(* PLC project FiveDofPlatform_error_diag.import.xml, CODESYS CODESYS V3.5 SP20 Patch 4 *)
(* stored: creationDateTime 2026-08-01T11:31:50, modificationDateTime 2026-08-01T11:31:50 *)

PROGRAM AxisStatusFeedback_PRG
  VAR
    fbStatusX : Sm3_Basic.MC_ReadStatus;
    fbAxisErrorX : Sm3_Basic.MC_ReadAxisError;
    fbStatusY : Sm3_Basic.MC_ReadStatus;
    fbAxisErrorY : Sm3_Basic.MC_ReadAxisError;
    fbStatusZ : Sm3_Basic.MC_ReadStatus;
    fbAxisErrorZ : Sm3_Basic.MC_ReadAxisError;
    fbStatusB : Sm3_Basic.MC_ReadStatus;
    fbAxisErrorB : Sm3_Basic.MC_ReadAxisError;
    fbStatusC : Sm3_Basic.MC_ReadStatus;
    fbAxisErrorC : Sm3_Basic.MC_ReadAxisError;
    wStatusX : WORD;
    wStatusY : WORD;
    wStatusZ : WORD;
    wStatusB : WORD;
    wStatusC : WORD;
    dwAxisErrorX : DWORD;
    dwAxisErrorY : DWORD;
    dwAxisErrorZ : DWORD;
    dwAxisErrorB : DWORD;
    dwAxisErrorC : DWORD;
    bStatusErrorX : BOOL;
    bStatusFBErrorX : BOOL;
    bAxisErrorX : BOOL;
    bSwEndSwitchX : BOOL;
    bStatusErrorY : BOOL;
    bStatusFBErrorY : BOOL;
    bAxisErrorY : BOOL;
    bSwEndSwitchY : BOOL;
    bStatusErrorZ : BOOL;
    bStatusFBErrorZ : BOOL;
    bAxisErrorZ : BOOL;
    bSwEndSwitchZ : BOOL;
    bStatusErrorB : BOOL;
    bStatusFBErrorB : BOOL;
    bAxisErrorB : BOOL;
    bSwEndSwitchB : BOOL;
    bStatusErrorC : BOOL;
    bStatusFBErrorC : BOOL;
    bAxisErrorC : BOOL;
    bSwEndSwitchC : BOOL;
    eStatusErrorX : SMC_ERROR;
    eAxisReadErrorX : SMC_ERROR;
    bAxisReadErrorX : BOOL;
    eStatusErrorY : SMC_ERROR;
    eAxisReadErrorY : SMC_ERROR;
    bAxisReadErrorY : BOOL;
    eStatusErrorZ : SMC_ERROR;
    eAxisReadErrorZ : SMC_ERROR;
    bAxisReadErrorZ : BOOL;
    eStatusErrorB : SMC_ERROR;
    eAxisReadErrorB : SMC_ERROR;
    bAxisReadErrorB : BOOL;
    eStatusErrorC : SMC_ERROR;
    eAxisReadErrorC : SMC_ERROR;
    bAxisReadErrorC : BOOL;
    wEnableMismatchFeedback : WORD;
    wStatusErrorFeedback : WORD;
    wAxisReadErrorFeedback : WORD;
    wStatusFBErrorFeedback : WORD;
  END_VAR

            
// 本程序只做反馈和诊断，不直接控制轴运动。
// [32] 五轴总使能命令。
// [33..37] 五轴状态字。
// [38..47] 五轴驱动 AxisErrorID，来自 MC_ReadAxisError.AxisErrorID。
// [48] 五轴 AxisEnable 请求反馈。
// [49..58] 五轴 MC_ReadStatus.ErrorID。
// [59..68] 五轴 MC_ReadAxisError.ErrorID。
// [69..78] 五轴 MC_Power.ErrorID，由各单轴程序写入。
// [79..83] 五轴 MC_Power 诊断字，bit0=Status，bit1=Error。
// [84] 诊断版本号，26081 表示 2026-08-01 诊断版已生效。
// [85] 使能请求 TRUE 但 MC_ReadStatus 仍 Disabled 的位图。
// [86] MC_ReadStatus.Error 位图。
// [87] MC_ReadAxisError.Error 位图。
// [88] MC_ReadStatus.FBErrorOccured 位图。

fbStatusX(
    Axis := AXIS_X,
    Enable := TRUE,
    Valid => ,
    Busy => ,
    Error => bStatusErrorX,
    ErrorID => eStatusErrorX,
    Disabled => ,
    Errorstop => ,
    Stopping => ,
    StandStill => ,
    DiscreteMotion => ,
    ContinuousMotion => ,
    SynchronizedMotion => ,
    Homing => ,
    ConstantVelocity => ,
    Accelerating => ,
    Decelerating => ,
    FBErrorOccured => bStatusFBErrorX,
);

// MC_ReadAxisError.AxisErrorID 只表示驱动轴本体错误号。
// 如果网线断开导致 MC_ReadAxisError 自己报 Error，错误号会写到 arReg_data[59..60]。
fbAxisErrorX(
    Axis := AXIS_X,
    Enable := TRUE,
    Valid => ,
    Busy => ,
    Error => bAxisReadErrorX,
    ErrorID => eAxisReadErrorX,
    AxisError => bAxisErrorX,
    AxisErrorID => dwAxisErrorX,
    SWEndSwitchActive => bSwEndSwitchX
);
IF NOT bAxisErrorX THEN
    // 没有驱动轴本体错误时清零 AxisErrorID，但不清零各功能块自己的 ErrorID。
    dwAxisErrorX := DWORD#0;
END_IF;

// 把 X 轴 BOOL 状态压缩成一个 WORD 状态字输出到 arReg_data[33]。
wStatusX := WORD#0;
IF fbStatusX.Disabled THEN wStatusX := wStatusX OR WORD#16#0001; END_IF;
IF fbStatusX.Errorstop THEN wStatusX := wStatusX OR WORD#16#0002; END_IF;
IF fbStatusX.Stopping THEN wStatusX := wStatusX OR WORD#16#0004; END_IF;
IF fbStatusX.StandStill THEN wStatusX := wStatusX OR WORD#16#0008; END_IF;
IF fbStatusX.DiscreteMotion THEN wStatusX := wStatusX OR WORD#16#0010; END_IF;
IF fbStatusX.ContinuousMotion THEN wStatusX := wStatusX OR WORD#16#0020; END_IF;
IF fbStatusX.SynchronizedMotion THEN wStatusX := wStatusX OR WORD#16#0040; END_IF;
IF fbStatusX.Homing THEN wStatusX := wStatusX OR WORD#16#0080; END_IF;
IF fbStatusX.ConstantVelocity THEN wStatusX := wStatusX OR WORD#16#0100; END_IF;
IF fbStatusX.Accelerating THEN wStatusX := wStatusX OR WORD#16#0200; END_IF;
IF fbStatusX.Decelerating THEN wStatusX := wStatusX OR WORD#16#0400; END_IF;
IF bStatusErrorX THEN wStatusX := wStatusX OR WORD#16#0800; END_IF;
IF bStatusFBErrorX THEN wStatusX := wStatusX OR WORD#16#1000; END_IF;
IF bAxisErrorX THEN wStatusX := wStatusX OR WORD#16#4000; END_IF;
IF bSwEndSwitchX THEN wStatusX := wStatusX OR WORD#16#8000; END_IF;
arReg_data[33] := WORD_TO_INT(wStatusX);

// arReg_data[38..39] 保存 X 轴驱动 AxisErrorID。
arReg_data[38] := WORD_TO_INT(DWORD_TO_WORD(dwAxisErrorX));
arReg_data[39] := WORD_TO_INT(DWORD_TO_WORD(SHR(dwAxisErrorX, 16)));

// arReg_data[49..50] 保存 X 轴 MC_ReadStatus.ErrorID。
arReg_data[49] := WORD_TO_INT(DWORD_TO_WORD(TO_DWORD(eStatusErrorX)));
arReg_data[50] := WORD_TO_INT(DWORD_TO_WORD(SHR(TO_DWORD(eStatusErrorX), 16)));

// arReg_data[59..60] 保存 X 轴 MC_ReadAxisError.ErrorID。
arReg_data[59] := WORD_TO_INT(DWORD_TO_WORD(TO_DWORD(eAxisReadErrorX)));
arReg_data[60] := WORD_TO_INT(DWORD_TO_WORD(SHR(TO_DWORD(eAxisReadErrorX), 16)));

fbStatusY(
    Axis := AXIS_Y,
    Enable := TRUE,
    Valid => ,
    Busy => ,
    Error => bStatusErrorY,
    ErrorID => eStatusErrorY,
    Disabled => ,
    Errorstop => ,
    Stopping => ,
    StandStill => ,
    DiscreteMotion => ,
    ContinuousMotion => ,
    SynchronizedMotion => ,
    Homing => ,
    ConstantVelocity => ,
    Accelerating => ,
    Decelerating => ,
    FBErrorOccured => bStatusFBErrorY,
);

// MC_ReadAxisError.AxisErrorID 只表示驱动轴本体错误号。
// 如果网线断开导致 MC_ReadAxisError 自己报 Error，错误号会写到 arReg_data[61..62]。
fbAxisErrorY(
    Axis := AXIS_Y,
    Enable := TRUE,
    Valid => ,
    Busy => ,
    Error => bAxisReadErrorY,
    ErrorID => eAxisReadErrorY,
    AxisError => bAxisErrorY,
    AxisErrorID => dwAxisErrorY,
    SWEndSwitchActive => bSwEndSwitchY
);
IF NOT bAxisErrorY THEN
    // 没有驱动轴本体错误时清零 AxisErrorID，但不清零各功能块自己的 ErrorID。
    dwAxisErrorY := DWORD#0;
END_IF;

// 把 Y 轴 BOOL 状态压缩成一个 WORD 状态字输出到 arReg_data[34]。
wStatusY := WORD#0;
IF fbStatusY.Disabled THEN wStatusY := wStatusY OR WORD#16#0001; END_IF;
IF fbStatusY.Errorstop THEN wStatusY := wStatusY OR WORD#16#0002; END_IF;
IF fbStatusY.Stopping THEN wStatusY := wStatusY OR WORD#16#0004; END_IF;
IF fbStatusY.StandStill THEN wStatusY := wStatusY OR WORD#16#0008; END_IF;
IF fbStatusY.DiscreteMotion THEN wStatusY := wStatusY OR WORD#16#0010; END_IF;
IF fbStatusY.ContinuousMotion THEN wStatusY := wStatusY OR WORD#16#0020; END_IF;
IF fbStatusY.SynchronizedMotion THEN wStatusY := wStatusY OR WORD#16#0040; END_IF;
IF fbStatusY.Homing THEN wStatusY := wStatusY OR WORD#16#0080; END_IF;
IF fbStatusY.ConstantVelocity THEN wStatusY := wStatusY OR WORD#16#0100; END_IF;
IF fbStatusY.Accelerating THEN wStatusY := wStatusY OR WORD#16#0200; END_IF;
IF fbStatusY.Decelerating THEN wStatusY := wStatusY OR WORD#16#0400; END_IF;
IF bStatusErrorY THEN wStatusY := wStatusY OR WORD#16#0800; END_IF;
IF bStatusFBErrorY THEN wStatusY := wStatusY OR WORD#16#1000; END_IF;
IF bAxisErrorY THEN wStatusY := wStatusY OR WORD#16#4000; END_IF;
IF bSwEndSwitchY THEN wStatusY := wStatusY OR WORD#16#8000; END_IF;
arReg_data[34] := WORD_TO_INT(wStatusY);

// arReg_data[40..41] 保存 Y 轴驱动 AxisErrorID。
arReg_data[40] := WORD_TO_INT(DWORD_TO_WORD(dwAxisErrorY));
arReg_data[41] := WORD_TO_INT(DWORD_TO_WORD(SHR(dwAxisErrorY, 16)));

// arReg_data[51..52] 保存 Y 轴 MC_ReadStatus.ErrorID。
arReg_data[51] := WORD_TO_INT(DWORD_TO_WORD(TO_DWORD(eStatusErrorY)));
arReg_data[52] := WORD_TO_INT(DWORD_TO_WORD(SHR(TO_DWORD(eStatusErrorY), 16)));

// arReg_data[61..62] 保存 Y 轴 MC_ReadAxisError.ErrorID。
arReg_data[61] := WORD_TO_INT(DWORD_TO_WORD(TO_DWORD(eAxisReadErrorY)));
arReg_data[62] := WORD_TO_INT(DWORD_TO_WORD(SHR(TO_DWORD(eAxisReadErrorY), 16)));

fbStatusZ(
    Axis := AXIS_Z,
    Enable := TRUE,
    Valid => ,
    Busy => ,
    Error => bStatusErrorZ,
    ErrorID => eStatusErrorZ,
    Disabled => ,
    Errorstop => ,
    Stopping => ,
    StandStill => ,
    DiscreteMotion => ,
    ContinuousMotion => ,
    SynchronizedMotion => ,
    Homing => ,
    ConstantVelocity => ,
    Accelerating => ,
    Decelerating => ,
    FBErrorOccured => bStatusFBErrorZ,
);

// MC_ReadAxisError.AxisErrorID 只表示驱动轴本体错误号。
// 如果网线断开导致 MC_ReadAxisError 自己报 Error，错误号会写到 arReg_data[63..64]。
fbAxisErrorZ(
    Axis := AXIS_Z,
    Enable := TRUE,
    Valid => ,
    Busy => ,
    Error => bAxisReadErrorZ,
    ErrorID => eAxisReadErrorZ,
    AxisError => bAxisErrorZ,
    AxisErrorID => dwAxisErrorZ,
    SWEndSwitchActive => bSwEndSwitchZ
);
IF NOT bAxisErrorZ THEN
    // 没有驱动轴本体错误时清零 AxisErrorID，但不清零各功能块自己的 ErrorID。
    dwAxisErrorZ := DWORD#0;
END_IF;

// 把 Z 轴 BOOL 状态压缩成一个 WORD 状态字输出到 arReg_data[35]。
wStatusZ := WORD#0;
IF fbStatusZ.Disabled THEN wStatusZ := wStatusZ OR WORD#16#0001; END_IF;
IF fbStatusZ.Errorstop THEN wStatusZ := wStatusZ OR WORD#16#0002; END_IF;
IF fbStatusZ.Stopping THEN wStatusZ := wStatusZ OR WORD#16#0004; END_IF;
IF fbStatusZ.StandStill THEN wStatusZ := wStatusZ OR WORD#16#0008; END_IF;
IF fbStatusZ.DiscreteMotion THEN wStatusZ := wStatusZ OR WORD#16#0010; END_IF;
IF fbStatusZ.ContinuousMotion THEN wStatusZ := wStatusZ OR WORD#16#0020; END_IF;
IF fbStatusZ.SynchronizedMotion THEN wStatusZ := wStatusZ OR WORD#16#0040; END_IF;
IF fbStatusZ.Homing THEN wStatusZ := wStatusZ OR WORD#16#0080; END_IF;
IF fbStatusZ.ConstantVelocity THEN wStatusZ := wStatusZ OR WORD#16#0100; END_IF;
IF fbStatusZ.Accelerating THEN wStatusZ := wStatusZ OR WORD#16#0200; END_IF;
IF fbStatusZ.Decelerating THEN wStatusZ := wStatusZ OR WORD#16#0400; END_IF;
IF bStatusErrorZ THEN wStatusZ := wStatusZ OR WORD#16#0800; END_IF;
IF bStatusFBErrorZ THEN wStatusZ := wStatusZ OR WORD#16#1000; END_IF;
IF bAxisErrorZ THEN wStatusZ := wStatusZ OR WORD#16#4000; END_IF;
IF bSwEndSwitchZ THEN wStatusZ := wStatusZ OR WORD#16#8000; END_IF;
arReg_data[35] := WORD_TO_INT(wStatusZ);

// arReg_data[42..43] 保存 Z 轴驱动 AxisErrorID。
arReg_data[42] := WORD_TO_INT(DWORD_TO_WORD(dwAxisErrorZ));
arReg_data[43] := WORD_TO_INT(DWORD_TO_WORD(SHR(dwAxisErrorZ, 16)));

// arReg_data[53..54] 保存 Z 轴 MC_ReadStatus.ErrorID。
arReg_data[53] := WORD_TO_INT(DWORD_TO_WORD(TO_DWORD(eStatusErrorZ)));
arReg_data[54] := WORD_TO_INT(DWORD_TO_WORD(SHR(TO_DWORD(eStatusErrorZ), 16)));

// arReg_data[63..64] 保存 Z 轴 MC_ReadAxisError.ErrorID。
arReg_data[63] := WORD_TO_INT(DWORD_TO_WORD(TO_DWORD(eAxisReadErrorZ)));
arReg_data[64] := WORD_TO_INT(DWORD_TO_WORD(SHR(TO_DWORD(eAxisReadErrorZ), 16)));

fbStatusB(
    Axis := AXIS_B,
    Enable := TRUE,
    Valid => ,
    Busy => ,
    Error => bStatusErrorB,
    ErrorID => eStatusErrorB,
    Disabled => ,
    Errorstop => ,
    Stopping => ,
    StandStill => ,
    DiscreteMotion => ,
    ContinuousMotion => ,
    SynchronizedMotion => ,
    Homing => ,
    ConstantVelocity => ,
    Accelerating => ,
    Decelerating => ,
    FBErrorOccured => bStatusFBErrorB,
);

// MC_ReadAxisError.AxisErrorID 只表示驱动轴本体错误号。
// 如果网线断开导致 MC_ReadAxisError 自己报 Error，错误号会写到 arReg_data[65..66]。
fbAxisErrorB(
    Axis := AXIS_B,
    Enable := TRUE,
    Valid => ,
    Busy => ,
    Error => bAxisReadErrorB,
    ErrorID => eAxisReadErrorB,
    AxisError => bAxisErrorB,
    AxisErrorID => dwAxisErrorB,
    SWEndSwitchActive => bSwEndSwitchB
);
IF NOT bAxisErrorB THEN
    // 没有驱动轴本体错误时清零 AxisErrorID，但不清零各功能块自己的 ErrorID。
    dwAxisErrorB := DWORD#0;
END_IF;

// 把 B 轴 BOOL 状态压缩成一个 WORD 状态字输出到 arReg_data[36]。
wStatusB := WORD#0;
IF fbStatusB.Disabled THEN wStatusB := wStatusB OR WORD#16#0001; END_IF;
IF fbStatusB.Errorstop THEN wStatusB := wStatusB OR WORD#16#0002; END_IF;
IF fbStatusB.Stopping THEN wStatusB := wStatusB OR WORD#16#0004; END_IF;
IF fbStatusB.StandStill THEN wStatusB := wStatusB OR WORD#16#0008; END_IF;
IF fbStatusB.DiscreteMotion THEN wStatusB := wStatusB OR WORD#16#0010; END_IF;
IF fbStatusB.ContinuousMotion THEN wStatusB := wStatusB OR WORD#16#0020; END_IF;
IF fbStatusB.SynchronizedMotion THEN wStatusB := wStatusB OR WORD#16#0040; END_IF;
IF fbStatusB.Homing THEN wStatusB := wStatusB OR WORD#16#0080; END_IF;
IF fbStatusB.ConstantVelocity THEN wStatusB := wStatusB OR WORD#16#0100; END_IF;
IF fbStatusB.Accelerating THEN wStatusB := wStatusB OR WORD#16#0200; END_IF;
IF fbStatusB.Decelerating THEN wStatusB := wStatusB OR WORD#16#0400; END_IF;
IF bStatusErrorB THEN wStatusB := wStatusB OR WORD#16#0800; END_IF;
IF bStatusFBErrorB THEN wStatusB := wStatusB OR WORD#16#1000; END_IF;
IF bAxisErrorB THEN wStatusB := wStatusB OR WORD#16#4000; END_IF;
IF bSwEndSwitchB THEN wStatusB := wStatusB OR WORD#16#8000; END_IF;
arReg_data[36] := WORD_TO_INT(wStatusB);

// arReg_data[44..45] 保存 B 轴驱动 AxisErrorID。
arReg_data[44] := WORD_TO_INT(DWORD_TO_WORD(dwAxisErrorB));
arReg_data[45] := WORD_TO_INT(DWORD_TO_WORD(SHR(dwAxisErrorB, 16)));

// arReg_data[55..56] 保存 B 轴 MC_ReadStatus.ErrorID。
arReg_data[55] := WORD_TO_INT(DWORD_TO_WORD(TO_DWORD(eStatusErrorB)));
arReg_data[56] := WORD_TO_INT(DWORD_TO_WORD(SHR(TO_DWORD(eStatusErrorB), 16)));

// arReg_data[65..66] 保存 B 轴 MC_ReadAxisError.ErrorID。
arReg_data[65] := WORD_TO_INT(DWORD_TO_WORD(TO_DWORD(eAxisReadErrorB)));
arReg_data[66] := WORD_TO_INT(DWORD_TO_WORD(SHR(TO_DWORD(eAxisReadErrorB), 16)));

fbStatusC(
    Axis := AXIS_C,
    Enable := TRUE,
    Valid => ,
    Busy => ,
    Error => bStatusErrorC,
    ErrorID => eStatusErrorC,
    Disabled => ,
    Errorstop => ,
    Stopping => ,
    StandStill => ,
    DiscreteMotion => ,
    ContinuousMotion => ,
    SynchronizedMotion => ,
    Homing => ,
    ConstantVelocity => ,
    Accelerating => ,
    Decelerating => ,
    FBErrorOccured => bStatusFBErrorC,
);

// MC_ReadAxisError.AxisErrorID 只表示驱动轴本体错误号。
// 如果网线断开导致 MC_ReadAxisError 自己报 Error，错误号会写到 arReg_data[67..68]。
fbAxisErrorC(
    Axis := AXIS_C,
    Enable := TRUE,
    Valid => ,
    Busy => ,
    Error => bAxisReadErrorC,
    ErrorID => eAxisReadErrorC,
    AxisError => bAxisErrorC,
    AxisErrorID => dwAxisErrorC,
    SWEndSwitchActive => bSwEndSwitchC
);
IF NOT bAxisErrorC THEN
    // 没有驱动轴本体错误时清零 AxisErrorID，但不清零各功能块自己的 ErrorID。
    dwAxisErrorC := DWORD#0;
END_IF;

// 把 C 轴 BOOL 状态压缩成一个 WORD 状态字输出到 arReg_data[37]。
wStatusC := WORD#0;
IF fbStatusC.Disabled THEN wStatusC := wStatusC OR WORD#16#0001; END_IF;
IF fbStatusC.Errorstop THEN wStatusC := wStatusC OR WORD#16#0002; END_IF;
IF fbStatusC.Stopping THEN wStatusC := wStatusC OR WORD#16#0004; END_IF;
IF fbStatusC.StandStill THEN wStatusC := wStatusC OR WORD#16#0008; END_IF;
IF fbStatusC.DiscreteMotion THEN wStatusC := wStatusC OR WORD#16#0010; END_IF;
IF fbStatusC.ContinuousMotion THEN wStatusC := wStatusC OR WORD#16#0020; END_IF;
IF fbStatusC.SynchronizedMotion THEN wStatusC := wStatusC OR WORD#16#0040; END_IF;
IF fbStatusC.Homing THEN wStatusC := wStatusC OR WORD#16#0080; END_IF;
IF fbStatusC.ConstantVelocity THEN wStatusC := wStatusC OR WORD#16#0100; END_IF;
IF fbStatusC.Accelerating THEN wStatusC := wStatusC OR WORD#16#0200; END_IF;
IF fbStatusC.Decelerating THEN wStatusC := wStatusC OR WORD#16#0400; END_IF;
IF bStatusErrorC THEN wStatusC := wStatusC OR WORD#16#0800; END_IF;
IF bStatusFBErrorC THEN wStatusC := wStatusC OR WORD#16#1000; END_IF;
IF bAxisErrorC THEN wStatusC := wStatusC OR WORD#16#4000; END_IF;
IF bSwEndSwitchC THEN wStatusC := wStatusC OR WORD#16#8000; END_IF;
arReg_data[37] := WORD_TO_INT(wStatusC);

// arReg_data[46..47] 保存 C 轴驱动 AxisErrorID。
arReg_data[46] := WORD_TO_INT(DWORD_TO_WORD(dwAxisErrorC));
arReg_data[47] := WORD_TO_INT(DWORD_TO_WORD(SHR(dwAxisErrorC, 16)));

// arReg_data[57..58] 保存 C 轴 MC_ReadStatus.ErrorID。
arReg_data[57] := WORD_TO_INT(DWORD_TO_WORD(TO_DWORD(eStatusErrorC)));
arReg_data[58] := WORD_TO_INT(DWORD_TO_WORD(SHR(TO_DWORD(eStatusErrorC), 16)));

// arReg_data[67..68] 保存 C 轴 MC_ReadAxisError.ErrorID。
arReg_data[67] := WORD_TO_INT(DWORD_TO_WORD(TO_DWORD(eAxisReadErrorC)));
arReg_data[68] := WORD_TO_INT(DWORD_TO_WORD(SHR(TO_DWORD(eAxisReadErrorC), 16)));

// 诊断版本号，Python 可用它判断 [49..88] 是否已由新版 PLC 代码写入。
arReg_data[84] := 26081;

// 使能请求不一致：AxisEnable 请求为 TRUE，但 MC_ReadStatus 仍显示 Disabled。
wEnableMismatchFeedback := WORD#0;
IF GVL.Axes[1].AxisEnable AND fbStatusX.Disabled THEN wEnableMismatchFeedback := wEnableMismatchFeedback OR WORD#16#0001; END_IF;
IF GVL.Axes[2].AxisEnable AND fbStatusY.Disabled THEN wEnableMismatchFeedback := wEnableMismatchFeedback OR WORD#16#0002; END_IF;
IF GVL.Axes[3].AxisEnable AND fbStatusZ.Disabled THEN wEnableMismatchFeedback := wEnableMismatchFeedback OR WORD#16#0004; END_IF;
IF GVL.Axes[4].AxisEnable AND fbStatusB.Disabled THEN wEnableMismatchFeedback := wEnableMismatchFeedback OR WORD#16#0008; END_IF;
IF GVL.Axes[5].AxisEnable AND fbStatusC.Disabled THEN wEnableMismatchFeedback := wEnableMismatchFeedback OR WORD#16#0010; END_IF;
arReg_data[85] := WORD_TO_INT(wEnableMismatchFeedback);

// 汇总功能块错误位，便于 Python 快速判断是哪一类诊断报错。
wStatusErrorFeedback := WORD#0;
IF bStatusErrorX THEN wStatusErrorFeedback := wStatusErrorFeedback OR WORD#16#0001; END_IF;
IF bStatusErrorY THEN wStatusErrorFeedback := wStatusErrorFeedback OR WORD#16#0002; END_IF;
IF bStatusErrorZ THEN wStatusErrorFeedback := wStatusErrorFeedback OR WORD#16#0004; END_IF;
IF bStatusErrorB THEN wStatusErrorFeedback := wStatusErrorFeedback OR WORD#16#0008; END_IF;
IF bStatusErrorC THEN wStatusErrorFeedback := wStatusErrorFeedback OR WORD#16#0010; END_IF;
arReg_data[86] := WORD_TO_INT(wStatusErrorFeedback);

wAxisReadErrorFeedback := WORD#0;
IF bAxisReadErrorX THEN wAxisReadErrorFeedback := wAxisReadErrorFeedback OR WORD#16#0001; END_IF;
IF bAxisReadErrorY THEN wAxisReadErrorFeedback := wAxisReadErrorFeedback OR WORD#16#0002; END_IF;
IF bAxisReadErrorZ THEN wAxisReadErrorFeedback := wAxisReadErrorFeedback OR WORD#16#0004; END_IF;
IF bAxisReadErrorB THEN wAxisReadErrorFeedback := wAxisReadErrorFeedback OR WORD#16#0008; END_IF;
IF bAxisReadErrorC THEN wAxisReadErrorFeedback := wAxisReadErrorFeedback OR WORD#16#0010; END_IF;
arReg_data[87] := WORD_TO_INT(wAxisReadErrorFeedback);

wStatusFBErrorFeedback := WORD#0;
IF bStatusFBErrorX THEN wStatusFBErrorFeedback := wStatusFBErrorFeedback OR WORD#16#0001; END_IF;
IF bStatusFBErrorY THEN wStatusFBErrorFeedback := wStatusFBErrorFeedback OR WORD#16#0002; END_IF;
IF bStatusFBErrorZ THEN wStatusFBErrorFeedback := wStatusFBErrorFeedback OR WORD#16#0004; END_IF;
IF bStatusFBErrorB THEN wStatusFBErrorFeedback := wStatusFBErrorFeedback OR WORD#16#0008; END_IF;
IF bStatusFBErrorC THEN wStatusFBErrorFeedback := wStatusFBErrorFeedback OR WORD#16#0010; END_IF;
arReg_data[88] := WORD_TO_INT(wStatusFBErrorFeedback);

          
END_PROGRAM

PROGRAM AXIS_X_PRG
  VAR
    伺服使能 : Sm3_Basic.MC_Power;  (* 轴功能块实例 *)
    伺服绝对位置执行 : Sm3_Basic.MC_MoveAbsolute;
    伺服实际位置 : Sm3_Basic.MC_ReadActualPosition;
    伺服停止 : Sm3_Basic.MC_Stop;
    伺服复位 : Sm3_Basic.MC_Reset;
    伺服状态 : Sm3_Basic.MC_ReadStatus;
    复位轴组 : Sm3_Basic.SMC3_ReinitDrive;
    当前位置 : LREAL;  (* 变量 *)
    轴组复位 : BOOL;
    目标位置 : LREAL;
    目标速度 : LREAL;
    伺服错误状态 : BOOL;
    轴使能状态 : BOOL;
    总线状态 : BOOL;
    复位触发 : R_TRIG;  (* 报警清除相关 *)
    复位请求 : BOOL;
    复位中 : BOOL;
    POS_DEAD_ZONE : REAL := 0.01;  (* 死区常量 *)
    move_trigger : R_TRIG;
    AXIS_X_EXCUSE : BOOL := FALSE;
    log_msg : STRING(100);
    bPowerErrorDiag : BOOL;
    ePowerErrorDiag : SMC_ERROR;
    wPowerDiag : WORD;
  END_VAR

                    //------------------------------------------------------------------
// Z 轴控制逻辑（简化版 - 仅上升沿触发）
//------------------------------------------------------------------

// 读取实际位置
伺服实际位置(
    Axis    := AXIS_X,
    Enable  := TRUE,
    Position=> 当前位置
);
GVL.Axes[1].ActualAngle := 当前位置;

// 读取轴状态
伺服状态(
    Axis    := AXIS_X,
    Enable  := TRUE,
    Valid   => ,
    Busy    => ,
    Error   => 伺服错误状态,
    ErrorID => ,
    Disabled=> 总线状态
);

// 轴使能控制
伺服使能(
    Axis               := AXIS_X,
    Enable             := TRUE,
    bRegulatorOn       := GVL.Axes[1].AxisEnable,
    bDriveStart        := GVL.Axes[1].AxisEnable,
    Status             => 轴使能状态,
    bRegulatorRealState=> ,
    bDriveStartRealState=> ,
    Busy               => ,
    Error              => bPowerErrorDiag,
    ErrorID            => ePowerErrorDiag
);


// arReg_data[69..70] 保存本轴 MC_Power.ErrorID。
// 拔网线、驱动掉线、电机线导致的上使能故障，常先从这里体现。
arReg_data[69] := WORD_TO_INT(DWORD_TO_WORD(TO_DWORD(ePowerErrorDiag)));
arReg_data[70] := WORD_TO_INT(DWORD_TO_WORD(SHR(TO_DWORD(ePowerErrorDiag), 16)));

// arReg_data[79] 保存本轴 MC_Power 诊断字：bit0=Status，bit1=Error。
wPowerDiag := WORD#0;
IF 轴使能状态 THEN wPowerDiag := wPowerDiag OR WORD#16#0001; END_IF;
IF bPowerErrorDiag THEN wPowerDiag := wPowerDiag OR WORD#16#0002; END_IF;
arReg_data[79] := WORD_TO_INT(wPowerDiag);

// 目标位置、速度赋值（来自全局变量）
目标位置 := GVL.Axes[1].TargetAngle;
目标速度 :=  GVL.Axes[1].TargetVel;

// ********** 核心：上升沿触发运动 **********
// 使用 R_TRIG 检测 need_move 的上升沿
move_trigger(CLK := GVL.Axes[1].NeedMoveAxis);
IF move_trigger.Q THEN
    AXIS_X_EXCUSE := TRUE;   // 产生一个扫描周期的脉冲
	log_msg := 'X-axis has been triggered';
// 	logfb(write:=TRUE,sFileTestString:=log_msg);
	AppendLog(log_msg);
ELSE
    AXIS_X_EXCUSE := FALSE;
END_IF

// 绝对定位指令
GVL.Axes[1].伺服绝对位置执行(
    Axis        := AXIS_X,
    Execute     := AXIS_X_EXCUSE,
    Position    := 目标位置,
    Velocity    := 目标速度,
    Acceleration:= 10000,//4000  //85000
    Deceleration:= 10000,//4000  //85000
    Jerk        := ,
    Direction   := ,
    BufferMode  := ,
    Done        => GVL.Axes[1].InitDone,
    Busy        => ,
    Active      => ,
    CommandAborted=> ,
    Error       => GVL.Axes[1].AxisError,
    ErrorID     =>
);

// 运动完成：清除 need_move 并通知状态机
IF  GVL.Axes[1].InitDone THEN
    GVL.Axes[1].NeedMoveAxis := FALSE;              // 清除运动请求
    GVL.Axes[1].AxisDone := TRUE;         // 通知状态机运动完成
	log_msg := 'X-Axis movement completed! ';
// 	logfb(write:=TRUE,sFileTestString:=log_msg);
// 	AppendLog(log_msg);
END_IF

// 复位功能块（保持不变）
伺服复位(
    Axis    := AXIS_X,
    Execute := 复位中 AND NOT 伺服复位.Done,
    Done    => ,
    Busy    => ,
    Error   => ,
    ErrorID =>
);

复位轴组(
    Axis      := AXIS_X,
    bExecute  := 伺服复位.Done,
    bVirtual  := FALSE,
    bDone     => ,
    bBusy     => ,
    bError    => ,
    nErrorID  =>
);

// 报警清除逻辑
复位触发(CLK := (伺服错误状态 OR 复位请求) AND NOT 复位中);
IF 复位触发.Q THEN
    复位中 := TRUE;
    复位请求 := FALSE;
END_IF

IF 伺服复位.Done THEN
    复位中 := FALSE;
END_IF
                  
END_PROGRAM

PROGRAM Axis_Y_PRG
  VAR
    伺服使能 : Sm3_Basic.MC_Power;  (* 轴功能块实例 *)
    伺服绝对位置执行 : Sm3_Basic.MC_MoveAbsolute;
    伺服实际位置 : Sm3_Basic.MC_ReadActualPosition;
    伺服停止 : Sm3_Basic.MC_Stop;
    伺服复位 : Sm3_Basic.MC_Reset;
    伺服状态 : Sm3_Basic.MC_ReadStatus;
    复位轴组 : Sm3_Basic.SMC3_ReinitDrive;
    当前位置 : LREAL;  (* 变量 *)
    轴组复位 : BOOL;
    目标位置 : LREAL;
    目标速度 : LREAL;
    伺服错误状态 : BOOL;
    轴使能状态 : BOOL;
    总线状态 : BOOL;
    复位触发 : R_TRIG;  (* 报警清除相关 *)
    复位请求 : BOOL;
    复位中 : BOOL;
    POS_DEAD_ZONE : REAL := 0.01;  (* 死区常量 *)
    伺服复位_Done : BOOL;
    debug_Done_Status : BOOL;  (* 在 AXIS_Y0_PRG 中添加 *)
    debug_KeepEnable : BOOL;
    move_trigger : R_TRIG;  (* 脉冲触发相关 *)
    AXIS_Y_EXCUSE : BOOL := FALSE;
    log_msg : STRING(100);
    bPowerErrorDiag : BOOL;
    ePowerErrorDiag : SMC_ERROR;
    wPowerDiag : WORD;
  END_VAR

                    //------------------------------------------------------------------
// Z 轴控制逻辑（简化版 - 仅上升沿触发）
//------------------------------------------------------------------

// 读取实际位置
伺服实际位置(
    Axis    := AXIS_Y,
    Enable  := TRUE,
    Position=> 当前位置
);
GVL.Axes[2].ActualAngle := 当前位置;

// 读取轴状态
伺服状态(
    Axis    := AXIS_Y,
    Enable  := TRUE,
    Valid   => ,
    Busy    => ,
    Error   => 伺服错误状态,
    ErrorID => ,
    Disabled=> 总线状态
);

// 轴使能控制
伺服使能(
    Axis               := AXIS_Y,
    Enable             := TRUE,
    bRegulatorOn       := GVL.Axes[2].AxisEnable,
    bDriveStart        := GVL.Axes[2].AxisEnable,
    Status             => 轴使能状态,
    bRegulatorRealState=> ,
    bDriveStartRealState=> ,
    Busy               => ,
    Error              => bPowerErrorDiag,
    ErrorID            => ePowerErrorDiag
);


// arReg_data[71..72] 保存本轴 MC_Power.ErrorID。
// 拔网线、驱动掉线、电机线导致的上使能故障，常先从这里体现。
arReg_data[71] := WORD_TO_INT(DWORD_TO_WORD(TO_DWORD(ePowerErrorDiag)));
arReg_data[72] := WORD_TO_INT(DWORD_TO_WORD(SHR(TO_DWORD(ePowerErrorDiag), 16)));

// arReg_data[80] 保存本轴 MC_Power 诊断字：bit0=Status，bit1=Error。
wPowerDiag := WORD#0;
IF 轴使能状态 THEN wPowerDiag := wPowerDiag OR WORD#16#0001; END_IF;
IF bPowerErrorDiag THEN wPowerDiag := wPowerDiag OR WORD#16#0002; END_IF;
arReg_data[80] := WORD_TO_INT(wPowerDiag);

// 目标位置、速度赋值（来自全局变量）
目标位置 := GVL.Axes[2].TargetAngle;
目标速度 :=  GVL.Axes[2].TargetVel;

// ********** 核心：上升沿触发运动 **********
// 使用 R_TRIG 检测 need_move 的上升沿
move_trigger(CLK := GVL.Axes[2].NeedMoveAxis);
IF move_trigger.Q THEN
    AXIS_Y_EXCUSE := TRUE;   // 产生一个扫描周期的脉冲
	log_msg := 'X-axis has been triggered';
// 	logfb(write:=TRUE,sFileTestString:=log_msg);
	AppendLog(log_msg);
ELSE
    AXIS_Y_EXCUSE := FALSE;
END_IF

// 绝对定位指令
GVL.Axes[2].伺服绝对位置执行(
    Axis        := AXIS_Y,
    Execute     := AXIS_Y_EXCUSE,
    Position    := 目标位置,
    Velocity    := 目标速度,
    Acceleration:= 10000,//4000  //85000
    Deceleration:= 10000,//4000  //85000
    Jerk        := ,
    Direction   := ,
    BufferMode  := ,
    Done        => GVL.Axes[2].InitDone,
    Busy        => ,
    Active      => ,
    CommandAborted=> ,
    Error       => GVL.Axes[2].AxisError,
    ErrorID     =>
);

// 运动完成：清除 need_move 并通知状态机
IF  GVL.Axes[2].InitDone THEN
    GVL.Axes[2].NeedMoveAxis := FALSE;              // 清除运动请求
    GVL.Axes[2].AxisDone := TRUE;         // 通知状态机运动完成
	log_msg := 'X-Axis movement completed! ';
// 	logfb(write:=TRUE,sFileTestString:=log_msg);
// 	AppendLog(log_msg);
END_IF

// 复位功能块（保持不变）
伺服复位(
    Axis    := AXIS_Y,
    Execute := 复位中 AND NOT 伺服复位.Done,
    Done    => ,
    Busy    => ,
    Error   => ,
    ErrorID =>
);

复位轴组(
    Axis      := AXIS_Y,
    bExecute  := 伺服复位.Done,
    bVirtual  := FALSE,
    bDone     => ,
    bBusy     => ,
    bError    => ,
    nErrorID  =>
);

// 报警清除逻辑
复位触发(CLK := (伺服错误状态 OR 复位请求) AND NOT 复位中);
IF 复位触发.Q THEN
    复位中 := TRUE;
    复位请求 := FALSE;
END_IF

IF 伺服复位.Done THEN
    复位中 := FALSE;
END_IF
                  
END_PROGRAM

PROGRAM AXIS_Z_PRG
  VAR
    伺服使能 : Sm3_Basic.MC_Power;  (* 轴功能块实例 *)
    伺服绝对位置执行 : Sm3_Basic.MC_MoveAbsolute;
    伺服实际位置 : Sm3_Basic.MC_ReadActualPosition;
    伺服停止 : Sm3_Basic.MC_Stop;
    伺服复位 : Sm3_Basic.MC_Reset;
    伺服状态 : Sm3_Basic.MC_ReadStatus;
    复位轴组 : Sm3_Basic.SMC3_ReinitDrive;
    当前位置 : LREAL;  (* 变量 *)
    轴组复位 : BOOL;
    目标位置 : LREAL;
    目标速度 : LREAL;
    伺服错误状态 : BOOL;
    轴使能状态 : BOOL;
    总线状态 : BOOL;
    复位触发 : R_TRIG;  (* 报警清除相关 *)
    复位请求 : BOOL;
    复位中 : BOOL;
    伺服复位_Done : BOOL;
    debug_Done_Status : BOOL;  (* 在 AXIS_Z_PRG 中添加 *)
    debug_KeepEnable : BOOL;
    move_trigger : R_TRIG;  (* 脉冲触发相关 *)
    AXIS_Z_EXCUSE : BOOL := FALSE;
    log_msg : STRING(100);
    bPowerErrorDiag : BOOL;
    ePowerErrorDiag : SMC_ERROR;
    wPowerDiag : WORD;
  END_VAR

                    //------------------------------------------------------------------
// Z 轴控制逻辑（简化版 - 仅上升沿触发）
//------------------------------------------------------------------

// 读取实际位置
伺服实际位置(
    Axis    := AXIS_Z,
    Enable  := TRUE,
    Position=> 当前位置
);
GVL.Axes[3].ActualAngle := 当前位置;

// 读取轴状态
伺服状态(
    Axis    := AXIS_Z,
    Enable  := TRUE,
    Valid   => ,
    Busy    => ,
    Error   => 伺服错误状态,
    ErrorID => ,
    Disabled=> 总线状态
);

// 轴使能控制
伺服使能(
    Axis               := AXIS_Z,
    Enable             := TRUE,
    bRegulatorOn       := GVL.Axes[3].AxisEnable,
    bDriveStart        := GVL.Axes[3].AxisEnable,
    Status             => 轴使能状态,
    bRegulatorRealState=> ,
    bDriveStartRealState=> ,
    Busy               => ,
    Error              => bPowerErrorDiag,
    ErrorID            => ePowerErrorDiag
);


// arReg_data[73..74] 保存本轴 MC_Power.ErrorID。
// 拔网线、驱动掉线、电机线导致的上使能故障，常先从这里体现。
arReg_data[73] := WORD_TO_INT(DWORD_TO_WORD(TO_DWORD(ePowerErrorDiag)));
arReg_data[74] := WORD_TO_INT(DWORD_TO_WORD(SHR(TO_DWORD(ePowerErrorDiag), 16)));

// arReg_data[81] 保存本轴 MC_Power 诊断字：bit0=Status，bit1=Error。
wPowerDiag := WORD#0;
IF 轴使能状态 THEN wPowerDiag := wPowerDiag OR WORD#16#0001; END_IF;
IF bPowerErrorDiag THEN wPowerDiag := wPowerDiag OR WORD#16#0002; END_IF;
arReg_data[81] := WORD_TO_INT(wPowerDiag);

// 目标位置、速度赋值（来自全局变量）
目标位置 := GVL.Axes[3].TargetAngle;
目标速度 :=  GVL.Axes[3].TargetVel;

// ********** 核心：上升沿触发运动 **********
// 使用 R_TRIG 检测 need_move 的上升沿
move_trigger(CLK := GVL.Axes[3].NeedMoveAxis);
IF move_trigger.Q THEN
    AXIS_Z_EXCUSE := TRUE;   // 产生一个扫描周期的脉冲
	log_msg := 'X-axis has been triggered';
// 	logfb(write:=TRUE,sFileTestString:=log_msg);
	AppendLog(log_msg);
ELSE
    AXIS_Z_EXCUSE := FALSE;
END_IF

// 绝对定位指令
GVL.Axes[3].伺服绝对位置执行(
    Axis        := AXIS_Z,
    Execute     := AXIS_Z_EXCUSE,
    Position    := 目标位置,
    Velocity    := 目标速度,
    Acceleration:= 10000,//4000  //85000
    Deceleration:= 10000,//4000  //85000
    Jerk        := ,
    Direction   := ,
    BufferMode  := ,
    Done        => GVL.Axes[3].InitDone,
    Busy        => ,
    Active      => ,
    CommandAborted=> ,
    Error       => GVL.Axes[3].AxisError,
    ErrorID     =>
);

// 运动完成：清除 need_move 并通知状态机
IF  GVL.Axes[3].InitDone THEN
    GVL.Axes[3].NeedMoveAxis := FALSE;              // 清除运动请求
    GVL.Axes[3].AxisDone := TRUE;         // 通知状态机运动完成
	log_msg := 'Z-Axis movement completed! ';
// 	logfb(write:=TRUE,sFileTestString:=log_msg);
// 	AppendLog(log_msg);
END_IF

// 复位功能块（保持不变）
伺服复位(
    Axis    := AXIS_Z,
    Execute := 复位中 AND NOT 伺服复位.Done,
    Done    => ,
    Busy    => ,
    Error   => ,
    ErrorID =>
);

复位轴组(
    Axis      := AXIS_Z,
    bExecute  := 伺服复位.Done,
    bVirtual  := FALSE,
    bDone     => ,
    bBusy     => ,
    bError    => ,
    nErrorID  =>
);

// 报警清除逻辑
复位触发(CLK := (伺服错误状态 OR 复位请求) AND NOT 复位中);
IF 复位触发.Q THEN
    复位中 := TRUE;
    复位请求 := FALSE;
END_IF

IF 伺服复位.Done THEN
    复位中 := FALSE;
END_IF
                  
END_PROGRAM

PROGRAM AXIS_B_PRG
  VAR
    伺服使能 : Sm3_Basic.MC_Power;  (* 轴功能块实例 *)
    伺服绝对位置执行 : Sm3_Basic.MC_MoveAbsolute;
    伺服实际位置 : Sm3_Basic.MC_ReadActualPosition;
    伺服停止 : Sm3_Basic.MC_Stop;
    伺服复位 : Sm3_Basic.MC_Reset;
    伺服状态 : Sm3_Basic.MC_ReadStatus;
    复位轴组 : Sm3_Basic.SMC3_ReinitDrive;
    当前位置 : LREAL;  (* 变量 *)
    轴组复位 : BOOL;
    目标位置 : LREAL;
    目标速度 : LREAL;
    伺服错误状态 : BOOL;
    轴使能状态 : BOOL;
    总线状态 : BOOL;
    复位触发 : R_TRIG;  (* 报警清除相关 *)
    复位请求 : BOOL;
    复位中 : BOOL;
    move_trigger : R_TRIG;
    AXIS_B_EXCUSE : BOOL := FALSE;
    log_msg : STRING(100);
    bPowerErrorDiag : BOOL;
    ePowerErrorDiag : SMC_ERROR;
    wPowerDiag : WORD;
  END_VAR

                    //------------------------------------------------------------------
// Z 轴控制逻辑（简化版 - 仅上升沿触发）
//------------------------------------------------------------------

// 读取实际位置
伺服实际位置(
    Axis    := AXIS_B,
    Enable  := TRUE,
    Position=> 当前位置
);
GVL.Axes[4].ActualAngle := 当前位置;

// 读取轴状态
伺服状态(
    Axis    := AXIS_B,
    Enable  := TRUE,
    Valid   => ,
    Busy    => ,
    Error   => 伺服错误状态,
    ErrorID => ,
    Disabled=> 总线状态
);

// 轴使能控制
伺服使能(
    Axis               := AXIS_B,
    Enable             := TRUE,
    bRegulatorOn       := GVL.Axes[4].AxisEnable,
    bDriveStart        := GVL.Axes[4].AxisEnable,
    Status             => 轴使能状态,
    bRegulatorRealState=> ,
    bDriveStartRealState=> ,
    Busy               => ,
    Error              => bPowerErrorDiag,
    ErrorID            => ePowerErrorDiag
);


// arReg_data[75..76] 保存本轴 MC_Power.ErrorID。
// 拔网线、驱动掉线、电机线导致的上使能故障，常先从这里体现。
arReg_data[75] := WORD_TO_INT(DWORD_TO_WORD(TO_DWORD(ePowerErrorDiag)));
arReg_data[76] := WORD_TO_INT(DWORD_TO_WORD(SHR(TO_DWORD(ePowerErrorDiag), 16)));

// arReg_data[82] 保存本轴 MC_Power 诊断字：bit0=Status，bit1=Error。
wPowerDiag := WORD#0;
IF 轴使能状态 THEN wPowerDiag := wPowerDiag OR WORD#16#0001; END_IF;
IF bPowerErrorDiag THEN wPowerDiag := wPowerDiag OR WORD#16#0002; END_IF;
arReg_data[82] := WORD_TO_INT(wPowerDiag);

// 目标位置、速度赋值（来自全局变量）
目标位置 := GVL.Axes[4].TargetAngle;
目标速度 :=  GVL.Axes[4].TargetVel;

// ********** 核心：上升沿触发运动 **********
// 使用 R_TRIG 检测 need_move 的上升沿
move_trigger(CLK := GVL.Axes[4].NeedMoveAxis);
IF move_trigger.Q THEN
    AXIS_B_EXCUSE := TRUE;   // 产生一个扫描周期的脉冲
	log_msg := 'X-axis has been triggered';
// 	logfb(write:=TRUE,sFileTestString:=log_msg);
	AppendLog(log_msg);
ELSE
    AXIS_B_EXCUSE := FALSE;
END_IF

// 绝对定位指令
GVL.Axes[4].伺服绝对位置执行(
    Axis        := AXIS_B,
    Execute     := AXIS_B_EXCUSE,
    Position    := 目标位置,
    Velocity    := 目标速度,
    Acceleration:= 10000,//4000  //85000
    Deceleration:= 10000,//4000  //85000
    Jerk        := ,
    Direction   := ,
    BufferMode  := ,
    Done        => GVL.Axes[4].InitDone,
    Busy        => ,
    Active      => ,
    CommandAborted=> ,
    Error       => GVL.Axes[4].AxisError,
    ErrorID     =>
);

// 运动完成：清除 need_move 并通知状态机
IF  GVL.Axes[4].InitDone THEN
    GVL.Axes[4].NeedMoveAxis := FALSE;              // 清除运动请求
    GVL.Axes[4].AxisDone := TRUE;         // 通知状态机运动完成
	log_msg := 'B-Axis movement completed! ';
// 	logfb(write:=TRUE,sFileTestString:=log_msg);
// 	AppendLog(log_msg);
END_IF

// 复位功能块（保持不变）
伺服复位(
    Axis    := AXIS_B,
    Execute := 复位中 AND NOT 伺服复位.Done,
    Done    => ,
    Busy    => ,
    Error   => ,
    ErrorID =>
);

复位轴组(
    Axis      := AXIS_B,
    bExecute  := 伺服复位.Done,
    bVirtual  := FALSE,
    bDone     => ,
    bBusy     => ,
    bError    => ,
    nErrorID  =>
);

// 报警清除逻辑
复位触发(CLK := (伺服错误状态 OR 复位请求) AND NOT 复位中);
IF 复位触发.Q THEN
    复位中 := TRUE;
    复位请求 := FALSE;
END_IF

IF 伺服复位.Done THEN
    复位中 := FALSE;
END_IF
                  
END_PROGRAM

PROGRAM AXIS_C_PRG
  VAR
    伺服使能 : Sm3_Basic.MC_Power;  (* 轴功能块实例 *)
    伺服绝对位置执行 : Sm3_Basic.MC_MoveAbsolute;
    伺服实际位置 : Sm3_Basic.MC_ReadActualPosition;
    伺服停止 : Sm3_Basic.MC_Stop;
    伺服复位 : Sm3_Basic.MC_Reset;
    伺服状态 : Sm3_Basic.MC_ReadStatus;
    复位轴组 : Sm3_Basic.SMC3_ReinitDrive;
    当前位置 : LREAL;  (* 变量 *)
    轴组复位 : BOOL;
    目标位置 : LREAL;
    目标速度 : LREAL;
    伺服错误状态 : BOOL;
    轴使能状态 : BOOL;
    总线状态 : BOOL;
    复位触发 : R_TRIG;  (* 报警清除相关 *)
    复位请求 : BOOL;
    复位中 : BOOL;
    POS_DEAD_ZONE : REAL := 0.01;  (* 死区常量 *)
    diff_old : BOOL := FALSE;  (* 上升沿检测 *)
    diff : BOOL;
    保持使能 : BOOL := FALSE;  (* 控制 MC_Power.Enable *)
    EnRise : R_TRIG;  (* 外部使能上升沿 *)
    PowerStatusRise : R_TRIG;  (* 轴使能状态上升沿 *)
    move_trigger : R_TRIG;
    AXIS_C_EXCUSE : BOOL := FALSE;
    AXIS_C_Done_Internal : BOOL;
    log_msg : STRING(100);
    bPowerErrorDiag : BOOL;
    ePowerErrorDiag : SMC_ERROR;
    wPowerDiag : WORD;
  END_VAR

                    //------------------------------------------------------------------
// Z 轴控制逻辑（简化版 - 仅上升沿触发）
//------------------------------------------------------------------

// 读取实际位置
伺服实际位置(
    Axis    := AXIS_C,
    Enable  := TRUE,
    Position=> 当前位置
);
GVL.Axes[5].ActualAngle := 当前位置;

// 读取轴状态
伺服状态(
    Axis    := AXIS_C,
    Enable  := TRUE,
    Valid   => ,
    Busy    => ,
    Error   => 伺服错误状态,
    ErrorID => ,
    Disabled=> 总线状态
);

// 轴使能控制
伺服使能(
    Axis               := AXIS_C,
    Enable             := TRUE,
    bRegulatorOn       := GVL.Axes[5].AxisEnable,
    bDriveStart        := GVL.Axes[5].AxisEnable,
    Status             => 轴使能状态,
    bRegulatorRealState=> ,
    bDriveStartRealState=> ,
    Busy               => ,
    Error              => bPowerErrorDiag,
    ErrorID            => ePowerErrorDiag
);


// arReg_data[77..78] 保存本轴 MC_Power.ErrorID。
// 拔网线、驱动掉线、电机线导致的上使能故障，常先从这里体现。
arReg_data[77] := WORD_TO_INT(DWORD_TO_WORD(TO_DWORD(ePowerErrorDiag)));
arReg_data[78] := WORD_TO_INT(DWORD_TO_WORD(SHR(TO_DWORD(ePowerErrorDiag), 16)));

// arReg_data[83] 保存本轴 MC_Power 诊断字：bit0=Status，bit1=Error。
wPowerDiag := WORD#0;
IF 轴使能状态 THEN wPowerDiag := wPowerDiag OR WORD#16#0001; END_IF;
IF bPowerErrorDiag THEN wPowerDiag := wPowerDiag OR WORD#16#0002; END_IF;
arReg_data[83] := WORD_TO_INT(wPowerDiag);

// 目标位置、速度赋值（来自全局变量）
目标位置 := GVL.Axes[5].TargetAngle;
目标速度 :=  GVL.Axes[5].TargetVel;

// ********** 核心：上升沿触发运动 **********
// 使用 R_TRIG 检测 need_move 的上升沿
move_trigger(CLK := GVL.Axes[5].NeedMoveAxis);
IF move_trigger.Q THEN
    AXIS_C_EXCUSE := TRUE;   // 产生一个扫描周期的脉冲
	log_msg := 'C-axis has been triggered';
// 	logfb(write:=TRUE,sFileTestString:=log_msg);
	AppendLog(log_msg);
ELSE
    AXIS_C_EXCUSE := FALSE;
END_IF

// 绝对定位指令
GVL.Axes[5].伺服绝对位置执行(
    Axis        := AXIS_C,
    Execute     := AXIS_C_EXCUSE,
    Position    := 目标位置,
    Velocity    := 目标速度,
    Acceleration:= 10000,//4000  //85000
    Deceleration:= 10000,//4000  //85000
    Jerk        := ,
    Direction   := ,
    BufferMode  := ,
    Done        => GVL.Axes[5].InitDone,
    Busy        => ,
    Active      => ,
    CommandAborted=> ,
    Error       => GVL.Axes[5].AxisError,
    ErrorID     =>
);

// 运动完成：清除 need_move 并通知状态机
IF  GVL.Axes[5].InitDone THEN
    GVL.Axes[5].NeedMoveAxis := FALSE;              // 清除运动请求
    GVL.Axes[5].AxisDone := TRUE;         // 通知状态机运动完成
	log_msg := 'B-Axis movement completed! ';
// 	logfb(write:=TRUE,sFileTestString:=log_msg);
// 	AppendLog(log_msg);
END_IF

// 复位功能块（保持不变）
伺服复位(
    Axis    := AXIS_C,
    Execute := 复位中 AND NOT 伺服复位.Done,
    Done    => ,
    Busy    => ,
    Error   => ,
    ErrorID =>
);

复位轴组(
    Axis      := AXIS_C,
    bExecute  := 伺服复位.Done,
    bVirtual  := FALSE,
    bDone     => ,
    bBusy     => ,
    bError    => ,
    nErrorID  =>
);

// 报警清除逻辑
复位触发(CLK := (伺服错误状态 OR 复位请求) AND NOT 复位中);
IF 复位触发.Q THEN
    复位中 := TRUE;
    复位请求 := FALSE;
END_IF

IF 伺服复位.Done THEN
    复位中 := FALSE;
END_IF
                  
END_PROGRAM

PROGRAM JogX
  VAR
    fbJogX : FB_ServoJog;
    xServoEnable : BOOL := TRUE;
  END_VAR

                    

 



 xJogMode[1] := (arReg_data[19] AND WORD#16#0001) <> WORD#0; // X
 
  // ================================
  // 5轴点动控制
  // ================================

  // 点动侧使能跟随 arReg_data[32] 解析后的 GVL.Axes[1].AxisEnable。
  // 五轴总关闭时，点动功能块不会继续用本地 TRUE 保持上使能。
  xServoEnable := GVL.Axes[1].AxisEnable;

  fbJogX(
      Axis := AXIS_X,
      xServoOn := xServoEnable,
      xReset := FALSE,
      xJogFwd := xJogFwd[1],
      xJogRev := xJogRev[1],
      xLimitFwd := FALSE,
      xLimitRev := FALSE,
      lrJogVel := 100.0,
      lrAcc := 100.0,
      lrDec := 200.0,
      lrJerk := 0.0
  );

                  
END_PROGRAM

PROGRAM JogY
  VAR
    fbJogX : FB_ServoJog;
    fbJogY : FB_ServoJog;
    fbJogZ : FB_ServoJog;
    fbJogB : FB_ServoJog;
    fbJogC : FB_ServoJog;
    xServoEnable : BOOL := TRUE;
  END_VAR

                    

 




  // ================================
  // 5轴点动控制
  // ================================


  // 点动侧使能跟随 arReg_data[32] 解析后的 GVL.Axes[2].AxisEnable。
  // 五轴总关闭时，点动功能块不会继续用本地 TRUE 保持上使能。
  xServoEnable := GVL.Axes[2].AxisEnable;

  fbJogY(
      Axis := AXIS_Y,
      xServoOn := xServoEnable,
      xReset := FALSE,
      xJogFwd := xJogFwd[2],
      xJogRev := xJogRev[2],
      xLimitFwd := FALSE,
      xLimitRev := FALSE,
      lrJogVel := 100.0,
      lrAcc := 100.0,
      lrDec := 200.0,
      lrJerk := 0.0
  );

 
                  
END_PROGRAM

PROGRAM JogZ
  VAR
    fbJogX : FB_ServoJog;
    fbJogY : FB_ServoJog;
    fbJogZ : FB_ServoJog;
    fbJogB : FB_ServoJog;
    fbJogC : FB_ServoJog;
    xServoEnable : BOOL := TRUE;
  END_VAR

                    

 




  // ================================
  // 5轴点动控制
  // ================================

  

  // 点动侧使能跟随 arReg_data[32] 解析后的 GVL.Axes[3].AxisEnable。
  // 五轴总关闭时，点动功能块不会继续用本地 TRUE 保持上使能。
  xServoEnable := GVL.Axes[3].AxisEnable;

  fbJogZ(
      Axis := AXIS_Z,
      xServoOn := xServoEnable,
      xReset := FALSE,
      xJogFwd := xJogFwd[3],
      xJogRev := xJogRev[3],
      xLimitFwd := FALSE,
      xLimitRev := FALSE,
      lrJogVel := 100.0,
      lrAcc := 100.0,
      lrDec := 200.0,
      lrJerk := 0.0
  );

 
                  
END_PROGRAM

PROGRAM JogB
  VAR
    fbJogX : FB_ServoJog;
    fbJogY : FB_ServoJog;
    fbJogZ : FB_ServoJog;
    fbJogB : FB_ServoJog;
    fbJogC : FB_ServoJog;
    xServoEnable : BOOL := TRUE;
  END_VAR

                    

 




  // ================================
  // 5轴点动控制
  // ================================

  
  // 点动侧使能跟随 arReg_data[32] 解析后的 GVL.Axes[4].AxisEnable。
  // 五轴总关闭时，点动功能块不会继续用本地 TRUE 保持上使能。
  xServoEnable := GVL.Axes[4].AxisEnable;

  fbJogB(
      Axis := AXIS_B,
      xServoOn := xServoEnable,
      xReset := FALSE,
      xJogFwd := xJogFwd[4],
      xJogRev := xJogRev[4],
      xLimitFwd := FALSE,
      xLimitRev := FALSE,
      lrJogVel := 100.0,
      lrAcc := 100.0,
      lrDec := 200.0,
      lrJerk := 0.0
  );

 
                  
END_PROGRAM

PROGRAM JogC
  VAR
    fbJogX : FB_ServoJog;
    fbJogY : FB_ServoJog;
    fbJogZ : FB_ServoJog;
    fbJogB : FB_ServoJog;
    fbJogC : FB_ServoJog;
    xServoEnable : BOOL := TRUE;
  END_VAR

                    

 




  // ================================
  // 5轴点动控制
  // ================================

  // 点动侧使能跟随 arReg_data[32] 解析后的 GVL.Axes[5].AxisEnable。
  // 五轴总关闭时，点动功能块不会继续用本地 TRUE 保持上使能。
  xServoEnable := GVL.Axes[5].AxisEnable;

  fbJogC(
      Axis := AXIS_C,
      xServoOn := xServoEnable,
      xReset := FALSE,
      xJogFwd := xJogFwd[5],
      xJogRev := xJogRev[5],
      xLimitFwd := FALSE,
      xLimitRev := FALSE,
      lrJogVel := 100.0,
      lrAcc := 100.0,
      lrDec := 200.0,
      lrJerk := 0.0
  );
                  
END_PROGRAM

CONFIGURATION Device
  RESOURCE Application ON PLC
    TASK MainTask(INTERVAL := T#5ms, PRIORITY := 1);
    PROGRAM AxisEnableControl_PRG WITH MainTask : AxisEnableControl_PRG;
    PROGRAM JogX WITH MainTask : JogX;
    PROGRAM JogY WITH MainTask : JogY;
    PROGRAM JogZ WITH MainTask : JogZ;
    PROGRAM JogB WITH MainTask : JogB;
    PROGRAM JogC WITH MainTask : JogC;
    PROGRAM AXIS_X_PRG WITH MainTask : AXIS_X_PRG;
    PROGRAM Axis_Y_PRG WITH MainTask : Axis_Y_PRG;
    PROGRAM AXIS_Z_PRG WITH MainTask : AXIS_Z_PRG;
    PROGRAM AXIS_B_PRG WITH MainTask : AXIS_B_PRG;
    PROGRAM AXIS_C_PRG WITH MainTask : AXIS_C_PRG;
    PROGRAM FiveDOF_Platform_PRG WITH MainTask : FiveDOF_Platform_PRG;
    PROGRAM LogConsumer WITH MainTask : LogConsumer;
    PROGRAM PLC_PRG WITH MainTask : PLC_PRG;
    PROGRAM AxisStatusFeedback_PRG WITH MainTask : AxisStatusFeedback_PRG;
    PROGRAM ModbusTcpSlave WITH MainTask : ModbusTcpSlave;
  END_RESOURCE
END_CONFIGURATION
